TYPE ST_EL3446_MUX_REAL :
STRUCT
    nSelector : UINT := E_EL3446_Phase.Error_INDEX_Not_Valid;
    fValueRef : REFERENCE TO REAL;
END_STRUCT
END_TYPE

(* stored: Version 1.1.0.1, ProductVersion 3.1.4024.12
   DUT ST_EL3446_MUX_REAL: Id {f9edd503-af32-401f-9f0d-b38c5e4f8d87} *)
